// TwinCAT 3 PLC project RetentiveTimerUnitTest
// ProgramVersion: 3.1.4023.0
// libraries:
//   Retentive Timers, * (FisoThemes&Runtimevic)
//   Tc2_Standard, * (Beckhoff Automation GmbH)
//   Tc2_System, * (Beckhoff Automation GmbH)
//   Tc3_Module, * (Beckhoff Automation GmbH)
// project tree:
//   / PlcTask.TcTTO
//   POUs/ FB_A.TcPOU, FB_B.TcPOU, MAIN.TcPOU
// (motion and I/O tree: see PLC project retentivetimers)
// real-time tasks:
//   TASK PlcTask: cycle T#10ms, priority 20, ADS port 350
//   TASK PlcTask1: cycle T#10ms, priority 21, ADS port 351
//   TASK PlcTask2: cycle T#10ms, priority 22, ADS port 352

CONFIGURATION RetentiveTimerUnitTest
    RESOURCE PLC ON TwinCAT3
        TASK PlcTask(INTERVAL := T#10ms, PRIORITY := 22);
        PROGRAM MAIN WITH PlcTask : MAIN;
    END_RESOURCE
END_CONFIGURATION

// ---- POUs/MAIN.TcPOU
PROGRAM MAIN
VAR
	fbRStopwatch		: RTimers.Timer(E_timer_type.RStopwatch);
	
	fb_B : FB_B := (ppointer := __NEW(FB_A)); // try this instead
	sum :INT;
END_VAR

fbRStopwatch();

fb_B(sum=>sum );

END_PROGRAM

// ---- POUs/FB_B.TcPOU
FUNCTION_BLOCK FB_B
VAR_OUTPUT
	sum : INT;
END_VAR
VAR
	ppointer : POINTER TO FB_A;
END_VAR

sum := ppointer^.Sum(2,67);

END_FUNCTION_BLOCK

// ---- POUs/FB_A.TcPOU
{attribute 'enable_dynamic_creation'}
FUNCTION_BLOCK FB_A
VAR
	value : BOOL;
	value2 : REAL := 42;
END_VAR

METHOD Sum : INT
VAR_INPUT
	value1 : INT;
	value2: INT;
END_VAR
Sum := value1 + value2;
END_METHOD

END_FUNCTION_BLOCK
